// TIA Portal V20 export
DATA_BLOCK "Tippler_DB"   // DB400
// stored: AutoNumber false, InstanceOfName Tippler, InstanceOfType FB
"Tippler"
   // VAR_INPUT
   //    Pallet_On_Tippler : Bool;
   //    iA1LowClamp_BasePos : Bool;
   //    iA1UpClamp_BasePos : Bool;
   //    iA2LowClamp_BasePos : Bool;
   //    iA2UpClamp_BasePos : Bool;
   //    iA1LowClamp_WorkPos : Bool;
   //    iA1UpClamp_WorkPos : Bool;
   //    iA2LowClamp_WorkPos : Bool;
   //    iA2UpClamp_WorkPos : Bool;
   //    iArm1_AngleValue : Int;
   //    iArm2_AngleValue : Int;
   //    iArm1_BasePos : Bool;
   //    iArm2_BasePos : Bool;
   //    HMI_Control : Bool;
   //    HMI_ButtonUp : Bool;
   //    HMI_ButtonDown : Bool;
   //    iButton_Down : Bool;
   //    iButton_Up : Bool;
   // END_VAR
   // VAR_OUTPUT
   //    Fq_Main_Valve_Arms : Bool;
   //    Fq_Main_Valve_Clamps : Bool;
   //    Fq_HydraulicUnit : Bool;
   //    qArm1 : Int;
   //    qArm2 : Int;
   //    qLowerClamps_Backward : Bool;
   //    qUpperClamps_Backward : Bool;
   //    qLowerClamps_Forward : Bool;
   //    qUpperClamps_Forward : Bool;
   // END_VAR
   // VAR
   //    Hydraulic_Ready { S7_SetPoint := 'True'} : TON_TIME;
   //    Hydraulic_Off { S7_SetPoint := 'True'} : TON_TIME;
   //    LowerClamps { S7_SetPoint := 'True'} : "Clamp";
   //    UpperClamps { S7_SetPoint := 'True'} : "Clamp";
   //    Arms { S7_SetPoint := 'True'} : "Arms";
   //    "Step" { S7_SetPoint := 'True'} : Int;
   //    ReqArmsDown : Bool;
   //    ReqArmsUp : Bool;
   //    Arms_workPos : Bool;
   //    Arms_basePos : Bool;
   //    Arms_clampsOperPos { S7_SetPoint := 'True'} : Bool;
   //    Tippler_maintenance { S7_SetPoint := 'True'} : "Tippler_maintenance";
   //    ButtonArmsDown { S7_SetPoint := 'True'} : Bool;
   //    ButtonArmsUp { S7_SetPoint := 'True'} : Bool;
   //    ReqLowerClampsClose : Bool;
   //    ReqUpperClampsClose : Bool;
   //    ReqLowerClampsOpen : Bool;
   //    ReqUpperClampsOpen : Bool;
   //    Timer_ClampsWorkPos { S7_SetPoint := 'True'} : TON_TIME;
   //    Timer_ClampsBasePos { S7_SetPoint := 'True'} : TON_TIME;
   //    Tippler_keep_down { S7_SetPoint := 'True'} : TP_TIME;
   //    N_Trig_Button_Down { S7_SetPoint := 'True'} : Bool;
   // END_VAR
BEGIN
END_DATA_BLOCK
